FUNCTION_BLOCK ConsoleControl
  (* Standard: 61499-2 *)
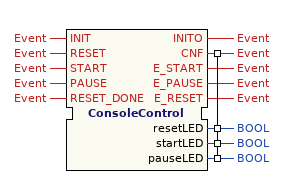
  EVENT_INPUT
    INIT;
    RESET;
    START;
    PAUSE;
    RESET_DONE;
  END_EVENT
  EVENT_OUTPUT
    INITO;
    CNF WITH resetLED, startLED, pauseLED;
    E_START;
    E_PAUSE;
    E_RESET;
  END_EVENT
  VAR_OUTPUT
    resetLED : BOOL;
    startLED : BOOL;
    pauseLED : BOOL;
  END_VAR
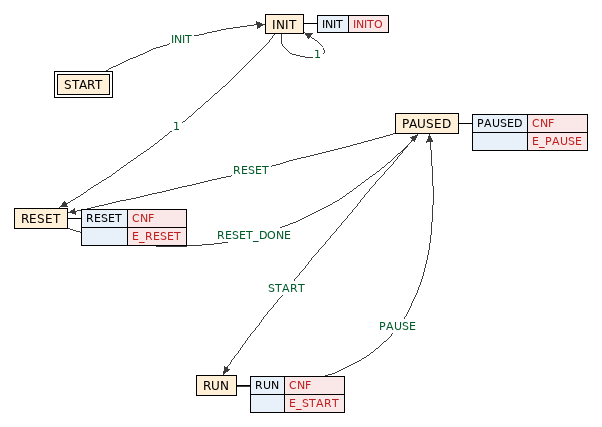
  EC_STATES
    START;
    INIT : INIT -> INITO;
    RESET : RESET -> CNF, -> E_RESET;
    PAUSED : PAUSED -> CNF, -> E_PAUSE;
    RUN : RUN -> CNF, -> E_START;
  END_STATES
  EC_TRANSITIONS
    START TO INIT := INIT;
    INIT TO RESET := 1;
    RESET TO PAUSED := RESET_DONE;
    PAUSED TO RUN := START;
    RUN TO PAUSED := PAUSE;
    PAUSED TO RESET := RESET;
    INIT TO INIT := 1;
  END_TRANSITIONS
  ALGORITHM INIT IN ST:
startLED := FALSE;&#10;pauseLED := FALSE;&#10;resetLED := TRUE;&#10;
  END_ALGORITHM
  ALGORITHM PAUSED IN ST:
startLED := FALSE;&#10;pauseLED := TRUE;&#10;resetLED := FALSE;&#10;
  END_ALGORITHM
  ALGORITHM RUN IN ST:
startLED := TRUE;&#10;pauseLED := FALSE;&#10;resetLED := FALSE;&#10;
  END_ALGORITHM
  ALGORITHM RESET IN ST:
startLED := FALSE;&#10;pauseLED := FALSE;&#10;resetLED := TRUE;&#10;
  END_ALGORITHM
END_FUNCTION_BLOCK
